FUNCTION_BLOCK ProgrammedOutput
VAR_INPUT
	
	
END_VAR
VAR_OUTPUT
END_VAR
VAR
	output AT%Q* : BOOL;
	isActivated : BOOL;
	
	duty : INT;
	
	dutyCounter : INT;	
	cycleCounter : INT;
END_VAR
VAR PERSISTENT
	//output duty cycle setting
	dutiesInPercentage : ARRAY[0..3] OF INT; //multiple setting
	cycleGoal : INT;
	baseTimer : TON;
END_VAR

IF baseTimer.Q AND isActivated THEN
	dutyCounter := dutyCounter+1;
END_IF

//output when in on duty cyle
output := isActivated AND (dutyCounter < duty) AND (cycleCounter<cycleGoal);

IF dutyCounter = duty THEN
	cycleCounter := cycleCounter +1;
END_IF

//rewind
IF dutyCounter >= 100 OR NOT isActivated THEN
	dutyCounter := 0;//reset
END_IF
IF cycleCounter >= cycleGoal OR NOT isActivated THEN
	cycleCounter := 0;//reset
END_IF

baseTimer(IN:= NOT baseTimer.Q, PT:= , Q=> , ET=> );

METHOD Activate : BOOL
VAR_INPUT
	set : int; // parameter set
END_VAR
duty := dutiesInPercentage[set];
isActivated := true;
END_METHOD

ACTION Deactivate:
isActivated := false;
END_ACTION

METHOD FB_init : BOOL
VAR_INPUT
	bInitRetains : BOOL; // if TRUE, the retain variables are initialized (warm start / cold start)
	bInCopyCode : BOOL;  // if TRUE, the instance afterwards gets moved into the copy code (online change)
END_VAR
IF bInitRetains THEN
	dutiesInPercentage[0] := 100;//always on
	dutiesInPercentage[1] := 75;//blink on
	dutiesInPercentage[2] := 50;//blink on
	dutiesInPercentage[3] := 25;//blink on
END_IF

baseTimer.PT := T#100MS; //default base
END_METHOD

END_FUNCTION_BLOCK

(* stored: Version 1.1.0.1, ProductVersion 3.1.4024.0
   POU ProgrammedOutput: Id {ba5e5d5f-de4b-4772-ba42-7511c7eb6187}, SpecialFunc None
   Method Activate: Id {0a0fe6dd-3262-4a80-8f95-cda1bc2fe9f0}
   Action Deactivate: Id {02b7f09e-4981-4ba7-b13f-358fe382a735}
   Method FB_init: Id {f41644d2-e25f-4243-9018-f07309d8edce} *)
